Universal Robots PolyScope program: Gripper signal timeout.urp

ProgramRoot directory=/home/ur/ursim-3.1/programs/Support site; kinematics=(a=[0, -0.425, -0.39225, 0, 0, 0], d=[0.08916, 0, 0, 0.10915, 0.09465, 0.0823], alpha=[1.5708, 0, 0, 1.5708, -1.5708, 0], deltaTheta=[0, 0, 0, 0, 0, 0], status=notInitialized); lastSavedInVersion=(project__name=Polyscope, major__version=3, minor__version=1, svn__revision=18024, build__date=Jul 07 2015, 15:18:49); name=Gripper signal timeout; programVersion=(project__name=Polyscope, major__version=3, minor__version=1, svn__revision=18024, build__date=Jul 07 2015, 15:18:49); robotEnvironmentFileName=default; serialNumberRobot=2015350001
  MainProgram cartesianAcceleration=1.2; cartesianSpeed=0.25; jointAcceleration=1.3962634015954636; jointSpeed=1.0471975511965976; sharedProcessMoveBlendRadius=0.025; motionType=JOINT_SPACE
    Comment commentString=Open gripper
    Set 
    If checkConditionInSeperateThread=true; expr=ExpressionIONode≟ False; type=IF_NODE
      Wait 
      Comment commentString=Gripper error
      Popup haltProgram=true; message=Gripper error; type=MESSAGE
    Comment commentString=Gripper OK
